{attribute 'qualified_only'}
{attribute 'strict'}
TYPE MF_SHAPE :
(
	Gaussian,
	Lshaped,
	Rshaped,
	Sshaped,
	Sigmoidal,
	Singleton,
	Trapeziodal,
	Triangular,
	Zshaped
);
END_TYPE

(* stored: Version 1.1.0.1, ProductVersion 3.1.4024.6
   DUT MF_SHAPE: Id {01523ae7-4e7d-4728-9512-5387b83507c9} *)
